// TIA Portal V17 export
// export: Created 2024-09-02T12:50:14.8224411Z, ExportSetting WithDefaults, DisplayName Totally Integrated Automation Portal, DisplayVersion V17, DisplayName TIA Portal Openness, DisplayVersion V17, DisplayName TIA Portal Version Control Interface, DisplayVersion V17, DisplayName STEP 7 Professional, DisplayVersion V17, DisplayName STEP 7 Safety, DisplayVersion V17, DisplayName WinCC Professional, DisplayVersion V17
DATA_BLOCK "AnwDB_ProcessData_FG02_OP70"   // DB501
TITLE = process data / Prozessdaten
{ S7_Optimized_Access := 'TRUE'; DB_Accessible_From_OPC_UA := 'FALSE' }
AUTHOR : VAF
FAMILY : PROZESS
NAME : PROZESS
VERSION : 0.1
// stored: AutoNumber false, DBAccessibleFromOPCUA false, IsOnlyStoredInLoadMemory false, IsRetainMemResEnabled false, IsWriteProtectedInAS false, MemoryReserve 100
   VAR RETAIN
      PROZESS { S7_SetPoint := 'True'} : Array[1..8] of "TypeProcessScreen";   // Werkerbild / worker's picture
      BEA : Array[1..8] of Struct   // Ergebnissdaten / Result data
         EBit : Array[1..32] of Struct   // Einzelbits / Individual bits
            Finished : Bool;   // Fertig / Finished
            OK : Bool;   // Ergebniss IO / Result OK
            NOK : Bool;   // Ergebniss NIO / Result NOK
            Started : Bool;
         END_STRUCT;
         Group : Array[0..3] of Struct   // Guppen / Group
            OK : Bool;   // Ergebniss IO / Result OK
            NOK : Bool;   // Ergebniss NIO / Result NOK
            Assembly_error_Activ : Bool;   // Montagefehler vorhanden / Mounting error present
            Deselection_Activ : Bool;   // Abwahl vorhanden / Choice available
            H_OK_Acitv : Bool;   // Hand-IO vorhanden / Hand-OK available
            Repeat_After_NOK : Bool;   // Wiederholen nach NIO aktiv / Repeat to NIO active
         END_STRUCT;
         Complete : Struct
            OK : Bool;   // Ergebniss IO / Result OK
            NOK : Bool;   // Ergebniss NIO / Result NOK
            Deselection_Active : Bool;   // Abwahl vorhanden / Choice available
            HOK_Active : Bool;   // Hand-IO vorhanden / Hand-OK available
            NA_Active : Bool;   // Nacharbeit vorhanden / Motor potentiometer up
            NOK_Active : Bool;   // NIO vorhanden / NIO present
            Repeat_After_NOK_Active : Bool;   // Wiederholen nach NIO aktiv / Repeat to NIO active
            NIO_Release_Active : Bool;   // NIO Entlassen aktiv / NIO Release active
            SG_Unlock : Bool;   // Schutztür entriegeln / UnBlocking the safety door
            SG_Lock : Bool;   // Schutztür verriegeln / Blocking the safety door
         END_STRUCT;
      END_STRUCT;
   END_VAR
BEGIN
END_DATA_BLOCK
